INTERFACE I_ContentVisitor

METHOD VisitContent
VAR_INPUT
	VisitingContent : I_Content;
END_VAR
END_METHOD

END_INTERFACE

(* stored: Version 1.1.0.1, ProductVersion 3.1.4024.12
   Itf I_ContentVisitor: Id {b904131c-36ac-0649-2fcc-4ca6fb3dfddf}
   Method VisitContent: Id {0eb13e90-f986-076c-04fb-a2abc7786a6c} *)
